// SIMATIC S7-200 SMART project (STEP 7-Micro/WIN SMART), CPU ST40

SYMBOL_TABLE Table 1
Start_switch     I0.0
Stop_switch      I0.1
Memory           M0.0
Solenoid_Valve   Q0.1
conveyer_belt    Q0.0
Sensor           I0.2
Timer1           T101
END_SYMBOL_TABLE

ORGANIZATION_BLOCK MAIN:OB1
TITLE=Program Comments
BEGIN
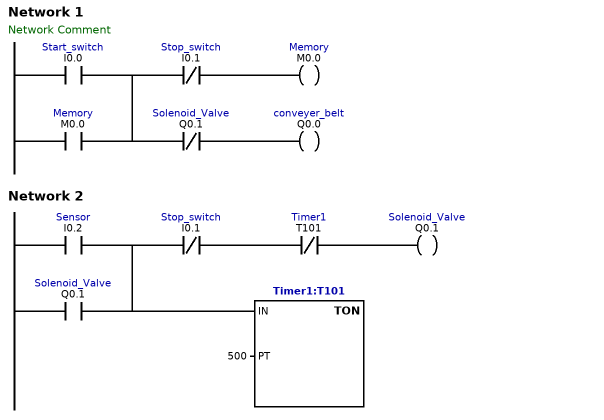
Network 1
// Network Comment
LD     Start_switch:I0.0
O      Memory:M0.0
LPS
AN     Stop_switch:I0.1
=      Memory:M0.0
LPP
AN     Solenoid_Valve:Q0.1
=      conveyer_belt:Q0.0
Network 2
// (network saved uncompiled; LAD cells follow)
// row 0: c0 -| |- Sensor:I0.2 v  c1 -|/|- Stop_switch:I0.1  c2 -|/|- Timer1:T101  c3 -( ) Solenoid_Valve:Q0.1
// row 1: c0 -| |- Solenoid_Valve:Q0.1 ^  c1 --  c2 [TON Timer1:T101 IN:=power@row1, PT:=500]
// row 2: c2 [box]
END_ORGANIZATION_BLOCK
